% RSLogix 500 project Project1.RSS, saved by version 8.30.00.16 %
PROJECT "UNTITLED"    % processor: Bul.1763 MicroLogix 1100 Series B %

PROGRAM FILES
  LAD 2 "MAIN"  3 rungs
  LAD 3 "DIGITAL IO"  5 rungs
  LAD 4 "CONTROLS"  11 rungs

DATA FILES
  O0 OUTPUT  4 elements
  I1 INPUT  6 elements
  S2 STATUS  66 elements
  B3 BINARY  1 elements
  T4 TIMER  5 elements
  C5 COUNTER  1 elements
  R6 CONTROL  1 elements
  N7 INTEGER  1 elements
  F8 FLOAT  1 elements

LADDER 2 "MAIN"
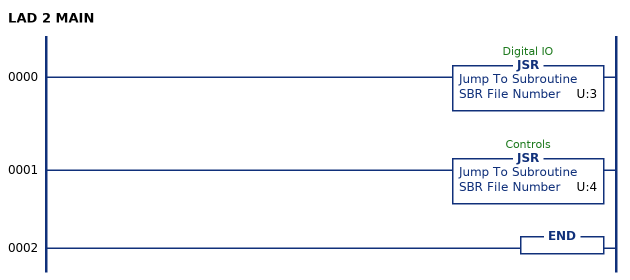
% Rung: 0 %
SOR JSR U:3 EOR
%   U:3  "Digital IO" %
% Rung: 1 %
SOR JSR U:4 EOR
%   U:4  "Controls" %
% Rung: 2 %
SOR END EOR

LADDER 3 "DIGITAL IO"
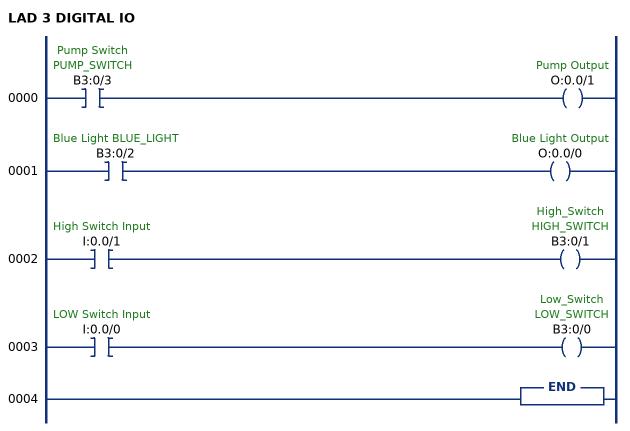
% Rung: 0 %
SOR XIC B3:0/3 OTE O:0.0/1 EOR
%   B3:0/3  PUMP_SWITCH  "Pump Switch" %
%   O:0.0/1  "Pump Output" %
% Rung: 1 %
SOR XIC B3:0/2 OTE O:0.0/0 EOR
%   B3:0/2  BLUE_LIGHT  "Blue Light" %
%   O:0.0/0  "Blue Light Output" %
% Rung: 2 %
SOR XIC I:0.0/1 OTE B3:0/1 EOR
%   I:0.0/1  "High Switch Input" %
%   B3:0/1  HIGH_SWITCH  "High_Switch" %
% Rung: 3 %
SOR XIC I:0.0/0 OTE B3:0/0 EOR
%   I:0.0/0  "LOW Switch Input" %
%   B3:0/0  LOW_SWITCH  "Low_Switch" %
% Rung: 4 %
SOR END EOR

LADDER 4 "CONTROLS"
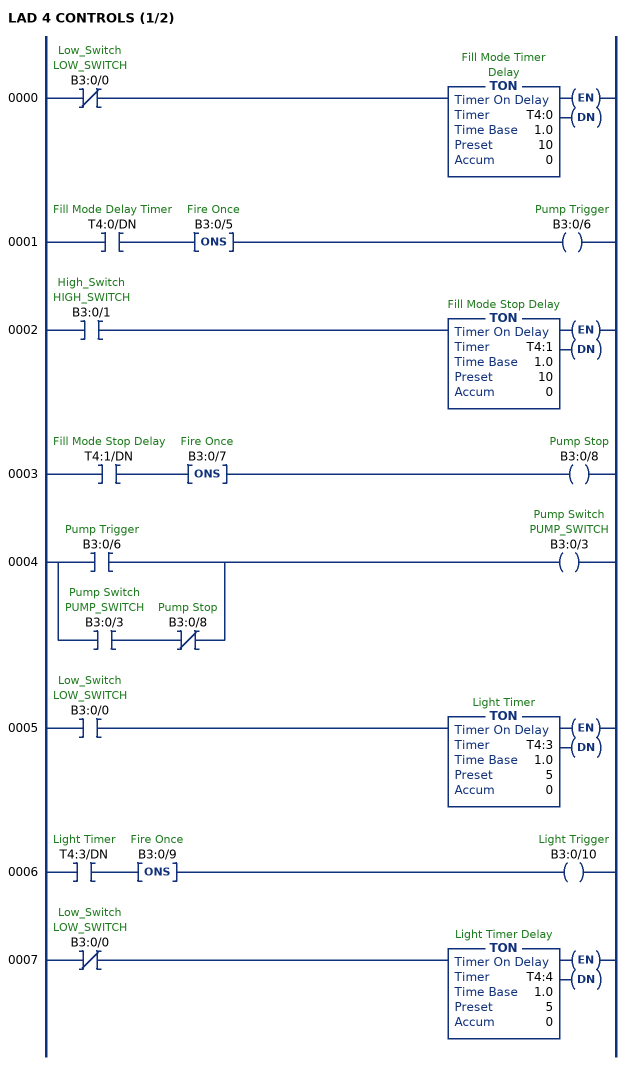
% Rung: 0 %
SOR XIO B3:0/0 TON T4:0 1.0 10 0 EOR
%   B3:0/0  LOW_SWITCH  "Low_Switch" %
%   T4:0  "Fill Mode Timer Delay" %
% Rung: 1 %
SOR XIC T4:0/DN ONS B3:0/5 OTE B3:0/6 EOR
%   T4:0/DN  "Fill Mode Delay Timer" %
%   B3:0/5  "Fire Once" %
%   B3:0/6  "Pump Trigger" %
% Rung: 2 %
SOR XIC B3:0/1 TON T4:1 1.0 10 0 EOR
%   B3:0/1  HIGH_SWITCH  "High_Switch" %
%   T4:1  "Fill Mode Stop Delay" %
% Rung: 3 %
SOR XIC T4:1/DN ONS B3:0/7 OTE B3:0/8 EOR
%   T4:1/DN  "Fill Mode Stop Delay" %
%   B3:0/7  "Fire Once" %
%   B3:0/8  "Pump Stop" %
% Rung: 4 %
SOR BST XIC B3:0/6 NXB XIC B3:0/3 XIO B3:0/8 BND OTE B3:0/3 EOR
%   B3:0/6  "Pump Trigger" %
%   B3:0/3  PUMP_SWITCH  "Pump Switch" %
%   B3:0/8  "Pump Stop" %
% Rung: 5 %
SOR XIC B3:0/0 TON T4:3 1.0 5 0 EOR
%   B3:0/0  LOW_SWITCH  "Low_Switch" %
%   T4:3  "Light Timer" %
% Rung: 6 %
SOR XIC T4:3/DN ONS B3:0/9 OTE B3:0/10 EOR
%   T4:3/DN  "Light Timer" %
%   B3:0/9  "Fire Once" %
%   B3:0/10  "Light Trigger" %
% Rung: 7 %
SOR XIO B3:0/0 TON T4:4 1.0 5 0 EOR
%   B3:0/0  LOW_SWITCH  "Low_Switch" %
%   T4:4  "Light Timer Delay" %

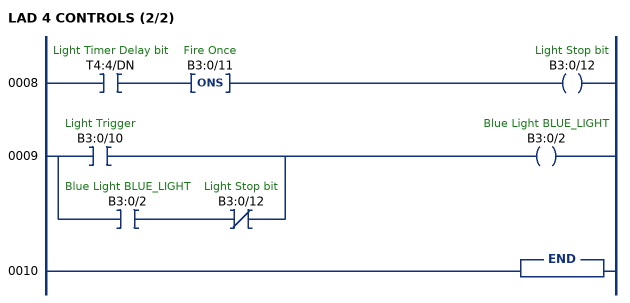
% Rung: 8 %
SOR XIC T4:4/DN ONS B3:0/11 OTE B3:0/12 EOR
%   T4:4/DN  "Light Timer Delay bit" %
%   B3:0/11  "Fire Once" %
%   B3:0/12  "Light Stop bit" %
% Rung: 9 %
SOR BST XIC B3:0/10 NXB XIC B3:0/2 XIO B3:0/12 BND OTE B3:0/2 EOR
%   B3:0/10  "Light Trigger" %
%   B3:0/2  BLUE_LIGHT  "Blue Light" %
%   B3:0/12  "Light Stop bit" %
% Rung: 10 %
SOR END EOR

OTHER DOCUMENTED ADDRESSES
  B3:0  "Turn On Light"
  B3:0/4  "Fill_Tank"
  T3:4  "Light OFF Timer"
  T3:4/DN  "Light Stop Delay"

DATA TABLE (non-zero values as saved)
DATA T4
% .PRE .ACC %
% T4:0 % 10 0
% T4:1 % 10 0
% T4:3 % 5 0
% T4:4 % 5 0
